# EPICS autosave request: iocBoot/iocUSB2408/auto_settings.req
file "USB2408_settings.req", P=USB2408:
